% RSLogix 500 project SWP.RSS, saved by version 8.30.00.16 %
PROJECT "UNTITLED"    % processor: Bul.1763 MicroLogix 1100 Series B %

PROGRAM FILES
  LAD 2   3 rungs

DATA FILES
  O0 OUTPUT  4 elements
  I1 INPUT  6 elements
  S2 STATUS  66 elements
  B3 BINARY  1 elements
  T4 TIMER  1 elements
  C5 COUNTER  1 elements
  R6 CONTROL  1 elements
  N7 INTEGER  2 elements
  F8 FLOAT  1 elements

LADDER 2
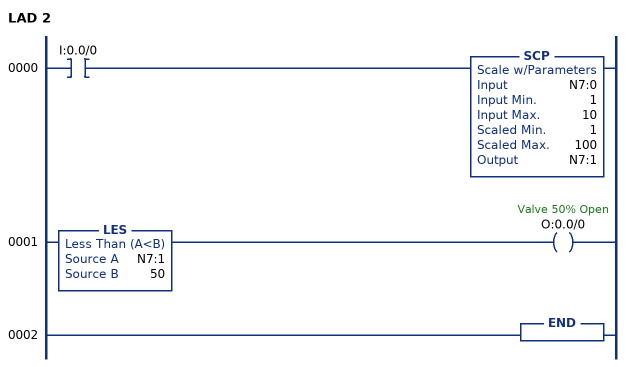
% Rung: 0 %  % edit flag set %
SOR XIC I:0.0/0 SCP N7:0 1 10 1 100 N7:1 EOR
% Rung: 1 %
SOR LES N7:1 50 OTE O:0.0/0 EOR
%   O:0.0/0  "Valve 50% Open" %
% Rung: 2 %
SOR END EOR
